// TIA Portal V20 export
TYPE "AnalogInDataHMI_DT"
   STRUCT
      ID_Measure : Int;
      CurrentValue : Real;
      TargetValue : Real;
      ThresholdAlarmMin : Real;
      ThresholdWarningMin : Real;
      ThresholdWarningMax : Real;
      ThresholdAlarmMax : Real;
      AxFactor { ExternalAccessible := 'False'; ExternalVisible := 'False'; ExternalWritable := 'False'} : Real := 1.0;   // A Factor Correction type y= Ax + B (A = 1 if no correction)
      BOffset { ExternalAccessible := 'False'; ExternalVisible := 'False'; ExternalWritable := 'False'} : Real;   // B Offset Correction type y= Ax + B (B = 0 if no correction)
      StartTime : Time;
      Update : Bool;
   END_STRUCT;
END_TYPE
